// TIA Portal V18 export
// export: Created 2026-06-08T16:04:38.1234394Z, ExportSetting WithDefaults, DisplayName Totally Integrated Automation Portal, DisplayVersion V18, DisplayName TIA Portal Openness, DisplayVersion V18, DisplayName TIA Portal Version Control Interface, DisplayVersion V18, DisplayName STEP 7 Professional, DisplayVersion V18, DisplayName STEP 7 Safety, DisplayVersion V18, DisplayName WinCC Professional, DisplayVersion V18
FUNCTION "FC_MANUAL_MODE" : Void   // FC1, LAD
{ S7_Optimized_Access := 'TRUE' }
VERSION : 0.1
// stored: AutoNumber true, IsIECCheckEnabled false, SetENOAutomatically false, UDAEnableTagReadback false
BEGIN

REGION Network 1: BĂNG TẢI
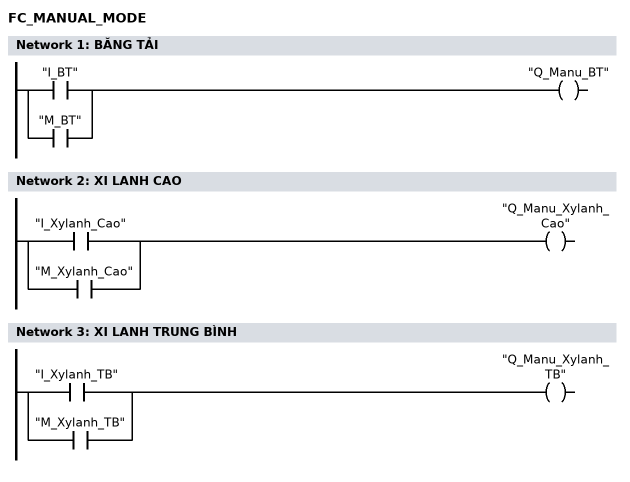
   RUNG wire#powerrail
      Contact( "I_BT" )
      wire#w1
      Coil( "Q_Manu_BT" )
   END_RUNG
   RUNG wire#powerrail
      Contact( "M_BT" )
   END_RUNG wire#w1
   // the same network as SCL:
   "Q_Manu_BT" := "I_BT" OR "M_BT";
END_REGION

REGION Network 2: XI LANH CAO
   RUNG wire#powerrail
      Contact( "I_Xylanh_Cao" )
      wire#w1
      Coil( "Q_Manu_Xylanh_Cao" )
   END_RUNG
   RUNG wire#powerrail
      Contact( "M_Xylanh_Cao" )
   END_RUNG wire#w1
   // the same network as SCL:
   "Q_Manu_Xylanh_Cao" := "I_Xylanh_Cao" OR "M_Xylanh_Cao";
END_REGION

REGION Network 3: XI LANH TRUNG BÌNH
   RUNG wire#powerrail
      Contact( "I_Xylanh_TB" )
      wire#w1
      Coil( "Q_Manu_Xylanh_TB" )
   END_RUNG
   RUNG wire#powerrail
      Contact( "M_Xylanh_TB" )
   END_RUNG wire#w1
   // the same network as SCL:
   "Q_Manu_Xylanh_TB" := "I_Xylanh_TB" OR "M_Xylanh_TB";
END_REGION
END_FUNCTION
